(*An interface describes the must have methods for a functionblock
	-now you know for sure that a block implementing this interface will have the methods described here
*) 
INTERFACE IOopExmpl

METHOD MustHaveMethod : BOOL
VAR_INPUT
	I:BOOL;
END_VAR
END_METHOD

END_INTERFACE

(* stored: Version 1.1.0.1
   Itf IOopExmpl: Id {8c04f71c-6e21-0b5c-368e-3e6351299a76}
   Method MustHaveMethod: Id {4c21514d-9d57-0f32-18b4-3eafb1df0e4e} *)
